FUNCTION Or3 : I_BoolValue
VAR_INPUT
	value1 : I_BoolValue;
	value2 : I_BoolValue;
	value3 : I_BoolValue;
END_VAR
VAR
	p : POINTER TO FB_BooleanExpression;
END_VAR

p := __NEW(FB_BooleanExpression);

p^.Op3(
	operator := E_BooleanOperator.ORop,
	value1 := value1,
	value2 := value2,
	value3 := value3
);

Or3 := p^;

END_FUNCTION

(* stored: Version 1.1.0.1
   POU Or3: Id {c72b0347-87bd-46ec-89a7-d2db3bc53b65}, SpecialFunc None *)
